// TIA Portal V20 export
// export: Created 2026-04-11T06:02:30.4980467Z, ExportSetting WithDefaults, DisplayName Totally Integrated Automation Portal, DisplayVersion V20, DisplayName TIA Portal Openness, DisplayVersion V20, DisplayName TIA Portal Version Control Interface, DisplayVersion V20, DisplayName STEP 7 Professional, DisplayVersion V20, DisplayName STEP 7 Safety, DisplayVersion V20, DisplayName WinCC Basic/Comfort/Advanced, DisplayVersion V20, DisplayName WinCC Unified, DisplayVersion V20
TYPE "udtHMI_HopperControl_Control"
// stored: IsFailsafeCompliant false
   STRUCT
      rLLAlarm { S7_SetPoint := 'True'} : Real;   // Bulk Tank Low Level SP
      rHLAlarm { S7_SetPoint := 'True'} : Real;   // Bulk Tank High Level SP
      rLLProcess { S7_SetPoint := 'True'} : Real;   // Bulk Tank Low Level SP
      rHLProcess { S7_SetPoint := 'True'} : Real;   // Bulk Tank High Level SP
      rTankCapacity { S7_SetPoint := 'True'} : Real;   // Bulk Tank Capacity
      bPB_ResetError : Bool;
      iMode : Int;   // Current mode, 1= Auto, 2 = Manual/Override
      rManualLevel : Real;   // Manual override value
   END_STRUCT;
END_TYPE
